FUNCTION_BLOCK FB_PowerMotorOn
VAR_INPUT
	
	bPowerOn			:BOOL;
	bPowerOff			:BOOL;
	bNegOn				:BOOL;
	bPosOn				:BOOL;
	pST_Axesfunctions 	:POINTER TO ARRAY[1..C_Max_AxesCount] OF ST_Axesfunctions;
	pST_AX5kFunctions	:POINTER TO ARRAY[1..C_Max_AxesCount] OF ST_AX5kFunctions;
	pAXIS_REF			:POINTER TO ARRAY[1..C_Max_AxesCount] OF AXIS_REF;
	pArrIgnoreEnableList:POINTER TO ARRAY[1..C_Max_AxesCount] OF BOOL;
	
	
END_VAR
VAR_OUTPUT
	Done				:BOOL;
END_VAR
VAR_IN_OUT
	Execute				:BOOL;
END_VAR

VAR_TEMP
	i: INT;
	check: BOOL;
END_VAR
VAR
	t1: TON;
	t2: Ton;
	p: INT;
END_VAR

t1(IN:=NOT t1.Q , PT:=T#1S , Q=> , ET=> );
t2(PT:=T#0.5S , Q=> , ET=> );

IF Execute THEN
	Done:=FALSE;
	t2(IN:=TRUE);
	FOR	i:= 1 TO 2 DO//C_Max_AxesCount
		IF NOT pArrIgnoreEnableList^[i] THEN			
			pST_Axesfunctions^[i].bAxReleaseNeg:= bNegOn;
			pST_Axesfunctions^[i].bAxReleasePos:= bPosOn;
			pST_Axesfunctions^[i].bMcReset:=TRUE;
			pST_AX5kFunctions^[i].bAxResetDrive:=TRUE;
			IF bPowerOn AND NOT bPowerOff THEN;
				IF prg_Call_Recipe_Slow.bAllRecipesLoaded THEN;
					pST_Axesfunctions^[i].bMcPower:=TRUE;
				ELSE;
					//Skip until all recipes will loaded
				END_IF
				
			ELSIF bPowerOff AND NOT bPowerOn THEN;
				pST_Axesfunctions^[i].bMcPower:=FALSE;
 			ELSE;
				fbPrintErrMessageByID(sModuleDescription:='VADIM',sActErrorID:='4568');
			END_IF
		END_IF
	END_FOR
	
END_IF

IF t2.Q THEN
	//IF NOT done THEN
		FOR	i:= 1 TO C_Max_AxesCount DO
			IF NOT pArrIgnoreEnableList^[i] THEN
				pST_Axesfunctions^[i].bMcReset:=FALSE;
				pST_AX5kFunctions^[i].bAxResetDrive:=FALSE;
			END_IF
		END_FOR
	//END_IF
	t2(IN:=FALSE);
END_IF

IF t1.Q THEN
	check:=TRUE;
	FOR	i:= 1 TO C_Max_AxesCount DO
		IF NOT pArrIgnoreEnableList^[i] THEN
			IF NOT pAXIS_REF^[i].Status.Operational THEN
				check:=FALSE;
			END_IF
		END_IF
	END_FOR
	Done:=check;
END_IF
Execute:=FALSE;
bPowerOn:=FALSE;
bPowerOff:=FALSE;

END_FUNCTION_BLOCK

(* stored: Version 1.1.0.1, ProductVersion 3.1.4024.11
   POU FB_PowerMotorOn: Id {3b3ba6c5-43da-4ccc-8747-9027dd49f298}, SpecialFunc None *)
